PROGRAM MAP_OUT
VAR


  uTransportState     : U_XTS_TRANSPORT_STATE;
  uStationState       : U_STATION_STATE;
END_VAR




  memcpy(ADR(uTransportState),  ADR(GVL_XTS.XtsTransportState),   SIZEOF(ST_XTS_TRANSPORT_STATE));
  memcpy(ADR(uStationState),    ADR(GVL_XTS.StationState),        SIZEOF(uStationState));

END_PROGRAM

(* stored: Version 1.1.0.1, ProductVersion 3.1.4024.12
   POU MAP_OUT: Id {c5b05d38-318e-436f-a847-8491a50e7418}, SpecialFunc None *)
